{attribute 'GeneratedUsingTerminal: EK1122-0000-0018'}
{attribute addProperty BoxType "EK1122-0000-0018"}
{attribute addProperty Id "Beckhoff_ELM35xxsub_EK1100EK1100_AB5A94672"}
{attribute addProperty CRC "3779840093"}
{attribute addProperty Size "2"}
TYPE Beckhoff_ELM35xxEK1122_E14BC85D EXTENDS EK1122_AB5A9467 :
STRUCT
	{attribute addProperty Name "Beckhoff_ELM35xxsub_EK1100"}
	{attribute addProperty PreviousPort "Beckhoff ELM35xxEK1122 : D"}
	Beckhoff_ELM35xxsub_EK1100 : EK1100_AB5A9467;
END_STRUCT
END_TYPE

(* stored: Version 1.2.0.0, ProductVersion 3.1.4024.9
   DUT Beckhoff_ELM35xxEK1122_E14BC85D: Id {5204ca32-5ba4-4e1d-a149-c82052836e82} *)
